PROGRAM GantryRobotMotion
VAR
	
	//Speed settings Adjustible from Visu
	MCJogVelocity		: LREAL := 100.0;
	MCAutoVelocity		: LREAL := 250.0;
	mxMCButtonManLowVelocity 	: BOOL;
	

	//Homing motion Settings
	MCHomingMode	: MC_HomingMode := MC_HomingMode.MC_DefaultHoming ;
	iMCXCaibratePos 	: INT := 8;
	iMCYCaibratePos 	: INT := 8;
	iMCZCaibratePos 	: INT := 8;

	//Manual motion Settings
	MCJogMode		: E_JogMode 	:= E_JogMode.MC_JOGMODE_CONTINOUS;
	MCJogAcceleration	: LREAL := 500.0;
	MCJogDeceleration	: LREAL := 1500.0;
	MCJogJerk			: LREAL := 800.0;
	
	//Auto Motion Settings
	MCAutoAcceleration	: LREAL := 500.0;
	MCAutoDeceleration	: LREAL := 500.0;
	MCAutoJerk			: LREAL := 500.0;
	
	
	//Safe Transport Position
	MCYSafePos : LREAL := 160.0;
	MCZLiftDist : LREAL := 50.0;


	//Connection NC to Physical Servo Drives
	MCXAxisRef: AXIS_REF;
	MCYAxisRef: AXIS_REF;
	MCZAxisRef: AXIS_REF;

	
	// Auto motion Settings
	MCBufferMode   	: MC_BufferMode := MC_BufferMode.MC_Aborting;	
	
	

	//General Condition flags
	mxGeneralCOntrolOk: BOOL;
	mxButtonGeneralControlOn: BOOL;
	mxButtonGeneralControlOff: BOOL;
	mxButtonStartAuto : BOOL;
	mxButtonStopAuto : BOOL;
	mxButtonAutoMode: BOOL;
	mxGeneralControlOn: BOOL;	
	mxManualMode: BOOL;	
	mxAutoMode: BOOL;
	mxLimSwOK: BOOL;
	mxMCPowerOn: BOOL;
	mxAxesStatusOk: BOOL;
	mxAutoOn: BOOL;
	fbTONpuls1: TON;
	fbTONpuls2: TON;
	mxControlOff: BOOL;
	
	//Motor Control Function Block
	//MC  Power
	fbMCXPower: MC_Power;	//X-Axis
	mxMCXButtonByPass: BOOL;
	mxMCXPowerOn: BOOL;	

	fbMCYPower: MC_Power;	//Y-Axis
	mxMCYButtonByPass: BOOL;
	mxMCYPowerOn: BOOL;	
	
	fbMCZPower: MC_Power;	//Z-Axis
	mxMCZButtonByPass: BOOL;
	mxMCZPowerOn: BOOL;	
	
	
	// MC Read Status
	fbMCXReadStatus	: MC_ReadStatus;
	MCXAxisStatus	: ST_AxisStatus;
	mxMCXAxisError	: BOOL;

	fbMCYReadStatus	: MC_ReadStatus;
	MCYAxisStatus	: ST_AxisStatus;
	mxMCYAxisError	: BOOL;

	fbMCZReadStatus	: MC_ReadStatus;
	MCZAxisStatus	: ST_AxisStatus;
	mxMCZAxisError	: BOOL;

	
	// MC Read Actual Position
	fbMCXReadActualPosition: MC_ReadActualPosition;
	fbMCYReadActualPosition: MC_ReadActualPosition;
	fbMCZReadActualPosition: MC_ReadActualPosition;
	MCActualPos: AbsPosition;	
		
	//MC Reset
	fbMCXReset: MC_Reset;	
	fbMCYReset: MC_Reset;	
	fbMCZReset: MC_Reset;	
	mxButtonResetError:BOOL;

	//MC Homing 
	fbMCXHome: MC_Home;			//X-axis
	mxMCXButtonHoming: BOOL;
	mxMCXHomingDone: BOOL;	
	
	fbMCYHome: MC_Home;			//Y-axis
	mxMCYButtonHoming: BOOL;
	mxMCYHomingDone: BOOL;	
	
	fbMCZHome: MC_Home;			//Z-axis
	mxMCZButtonHoming: BOOL;
	mxMCZHomingDone: BOOL;	
	mxHomingDone: BOOL;	
	
	//MC Jog
	fbMCXJog: MC_Jog;			//X-Axis
	mxMCXButtonJogFWD: BOOL;
	mxMCXButtonJogBWD: BOOL;
	
	fbMCYJog: MC_Jog;			//Y-Axis
	mxMCYButtonJogFWD: BOOL;
	mxMCYButtonJogBWD: BOOL;
	
	fbMCZJog: MC_Jog;			//Z-Axis
	mxMCZButtonJogFWD: BOOL;
	mxMCZButtonJogBWD: BOOL;
	
	
	//MC Move Absolute Position	(Auto Sequence)
	fbMCXMoveAbsolute: MC_MoveAbsolute;		//X-Axis
	mxMCXMoveAbs: BOOL;
	MCXMovAbsPos: LREAL;
	MCXMoveAbsVel: LREAL;
	MCXMoveAbsACC: LREAL;
	MCXMoveAbsDec: LREAL;
	MCXMoveAbsJerk: LREAL;
	mxMCXMoveAbsDone: BOOL;

	//MC Move Absolute Position
	fbMCYMoveAbsolute: MC_MoveAbsolute;  	//Y-Axis
	mxMCYMoveAbs: BOOL;
	MCYMovAbsPos: LREAL;
	MCYMoveAbsVel: LREAL;
	MCYMoveAbsACC: LREAL;
	MCYMoveAbsDec: LREAL;
	MCYMoveAbsJerk: LREAL;
	mxMCYMoveAbsDone: BOOL;
	
	fbMCXHalt: MC_Halt;
	fbMCYHalt: MC_Halt;
	fbMCZHalt: MC_Halt;
	

	//MC Move Absolute Position
	fbMCZMoveAbsolute: MC_MoveAbsolute;		//Z-Axis
	mxMCZMoveAbs: BOOL;
	MCZMovAbsPos: LREAL;
	MCZMoveAbsVel: LREAL;
	MCZMoveAbsACC: LREAL;
	MCZMoveAbsDec: LREAL;
	MCZMoveAbsJerk: LREAL;
	mxMCZMoveAbsDone: BOOL;
	
	//Modify Position
	ModPos	: AbsPosition;
	ModPosStation: INT := 1;
	ModPosLocation:INT := 1;
	mxButtonModPosExecute : BOOL;
	mxButtonSavePos : BOOL;
	fbTONButtonModPosExecute : TON;
	mxButtonReadFile: BOOL;
	mxReminderToSave : BOOL;
	
	
	// Gripper	
	mxTogleGripper : BOOL;
	fbTONGripperOn: TON;
	fbTONGripperOff: TON;	
	
	//Auto Sequence
	iSequence: INT; 
	arrAbsPosition: ARRAY[1..4, 1..9] OF AbsPosition;	//Station 100-400 Place 1 to 9
	mxButtonGoToModPos : BOOL;
	strStatusText : STRING;
	
	
	//File handling AbsPositions XYZ
	fbFileOpen    			: FB_FileOpen;
    fbFileRead              : FB_FileRead;
    fbFileWrite             : FB_FileWrite;
    fbFileClose             : FB_FileClose;    
	hFile                   : UINT   := 0;
	mxFileOpen				: BOOL;
	mxFileRead				: BOOL;	
	mxFileWrite				: BOOL;
	mxFileClose				: BOOL;
	nFileOpenMode			: DWORD;
	mxMemSavePos: BOOL;
	mxMemReadFile: BOOL;
	fbTONFileTime: TON;

END_VAR
VAR // added by the converter: edge detectors and wires of the graphical bodies
    _rt1, _rt2, _rt3, _rt4, _rt5, _rt6, _rt7 : R_TRIG;
END_VAR

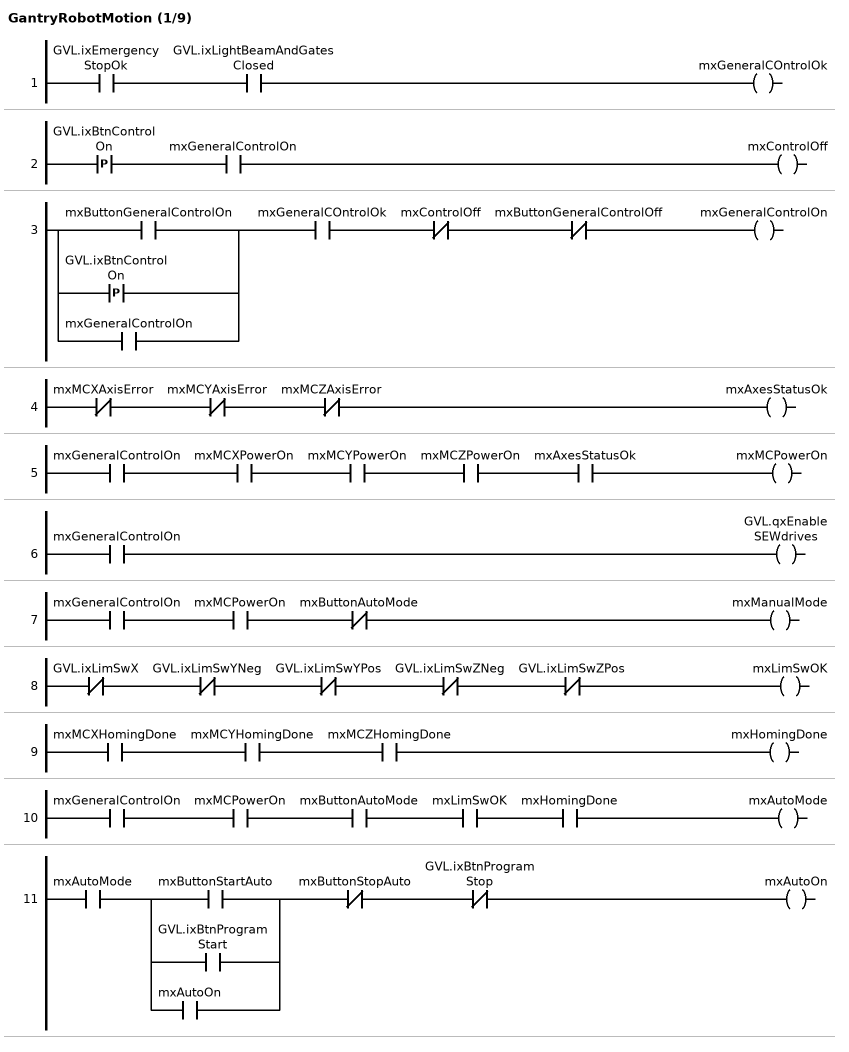
// NETWORK 1
mxGeneralCOntrolOk := GVL.ixEmergencyStopOk AND GVL.ixLightBeamAndGatesClosed;

// NETWORK 2
_rt1(CLK := GVL.ixBtnControlOn);
mxControlOff := _rt1.Q AND mxGeneralControlOn;

// NETWORK 3
_rt2(CLK := GVL.ixBtnControlOn);
mxGeneralControlOn := (mxButtonGeneralControlOn OR _rt2.Q OR mxGeneralControlOn) AND mxGeneralCOntrolOk AND NOT mxControlOff AND NOT mxButtonGeneralControlOff;

// NETWORK 4
mxAxesStatusOk := NOT mxMCXAxisError AND NOT mxMCYAxisError AND NOT mxMCZAxisError;

// NETWORK 5
mxMCPowerOn := mxGeneralControlOn AND mxMCXPowerOn AND mxMCYPowerOn AND mxMCZPowerOn AND mxAxesStatusOk;

// NETWORK 6
GVL.qxEnableSEWdrives := mxGeneralControlOn;

// NETWORK 7
mxManualMode := mxGeneralControlOn AND mxMCPowerOn AND NOT mxButtonAutoMode;

// NETWORK 8
mxLimSwOK := NOT GVL.ixLimSwX AND NOT GVL.ixLimSwYNeg AND NOT GVL.ixLimSwYPos AND NOT GVL.ixLimSwZNeg AND NOT GVL.ixLimSwZPos;

// NETWORK 9
mxHomingDone := mxMCXHomingDone AND mxMCYHomingDone AND mxMCZHomingDone;

// NETWORK 10
mxAutoMode := mxGeneralControlOn AND mxMCPowerOn AND mxButtonAutoMode AND mxLimSwOK AND mxHomingDone;

// NETWORK 11
mxAutoOn := mxAutoMode AND (mxButtonStartAuto OR GVL.ixBtnProgramStart OR mxAutoOn) AND NOT mxButtonStopAuto AND NOT GVL.ixBtnProgramStop;

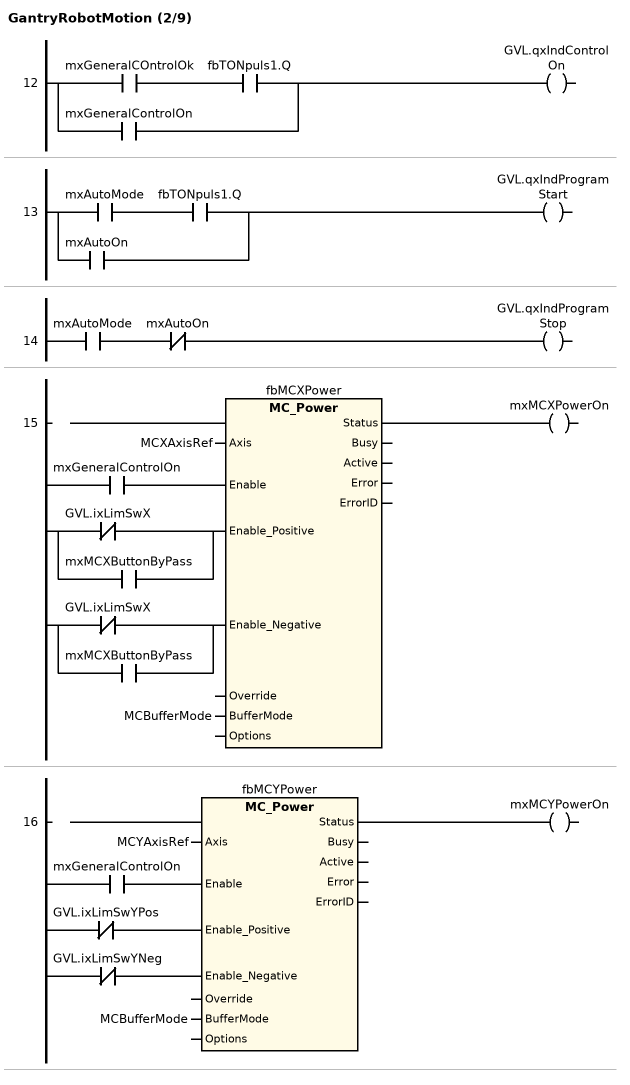
// NETWORK 12
GVL.qxIndControlOn := mxGeneralCOntrolOk AND fbTONpuls1.Q OR mxGeneralControlOn;

// NETWORK 13
GVL.qxIndProgramStart := mxAutoMode AND fbTONpuls1.Q OR mxAutoOn;

// NETWORK 14
GVL.qxIndProgramStop := mxAutoMode AND NOT mxAutoOn;

// NETWORK 15
fbMCXPower(
    Axis := MCXAxisRef,
    Enable := mxGeneralControlOn,
    Enable_Positive := NOT GVL.ixLimSwX OR mxMCXButtonByPass,
    Enable_Negative := NOT GVL.ixLimSwX OR mxMCXButtonByPass,
    BufferMode := MCBufferMode); // MC_Power
mxMCXPowerOn := fbMCXPower.Status;

// NETWORK 16
fbMCYPower(
    Axis := MCYAxisRef,
    Enable := mxGeneralControlOn,
    Enable_Positive := NOT GVL.ixLimSwYPos,
    Enable_Negative := NOT GVL.ixLimSwYNeg,
    BufferMode := MCBufferMode); // MC_Power
mxMCYPowerOn := fbMCYPower.Status;

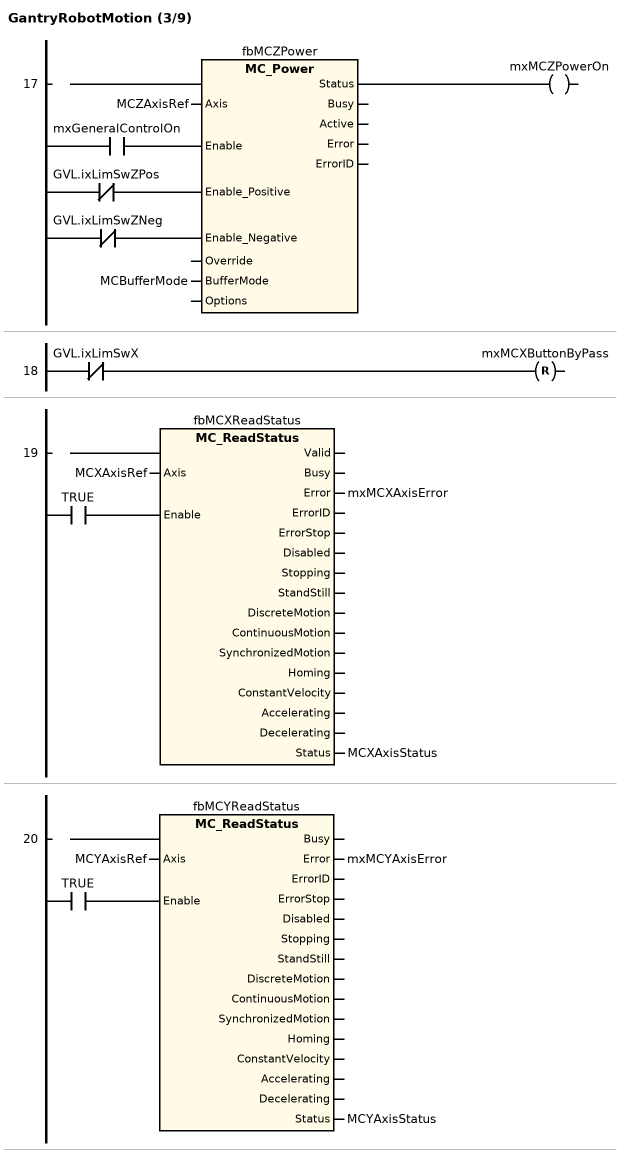
// NETWORK 17
fbMCZPower(
    Axis := MCZAxisRef,
    Enable := mxGeneralControlOn,
    Enable_Positive := NOT GVL.ixLimSwZPos,
    Enable_Negative := NOT GVL.ixLimSwZNeg,
    BufferMode := MCBufferMode); // MC_Power
mxMCZPowerOn := fbMCZPower.Status;

// NETWORK 18
mxMCXButtonByPass R= NOT GVL.ixLimSwX;

// NETWORK 19
fbMCXReadStatus(Axis := MCXAxisRef, Enable := TRUE, Error => mxMCXAxisError, Status => MCXAxisStatus); // MC_ReadStatus

// NETWORK 20
fbMCYReadStatus(Axis := MCYAxisRef, Enable := TRUE, Error => mxMCYAxisError, Status => MCYAxisStatus); // MC_ReadStatus

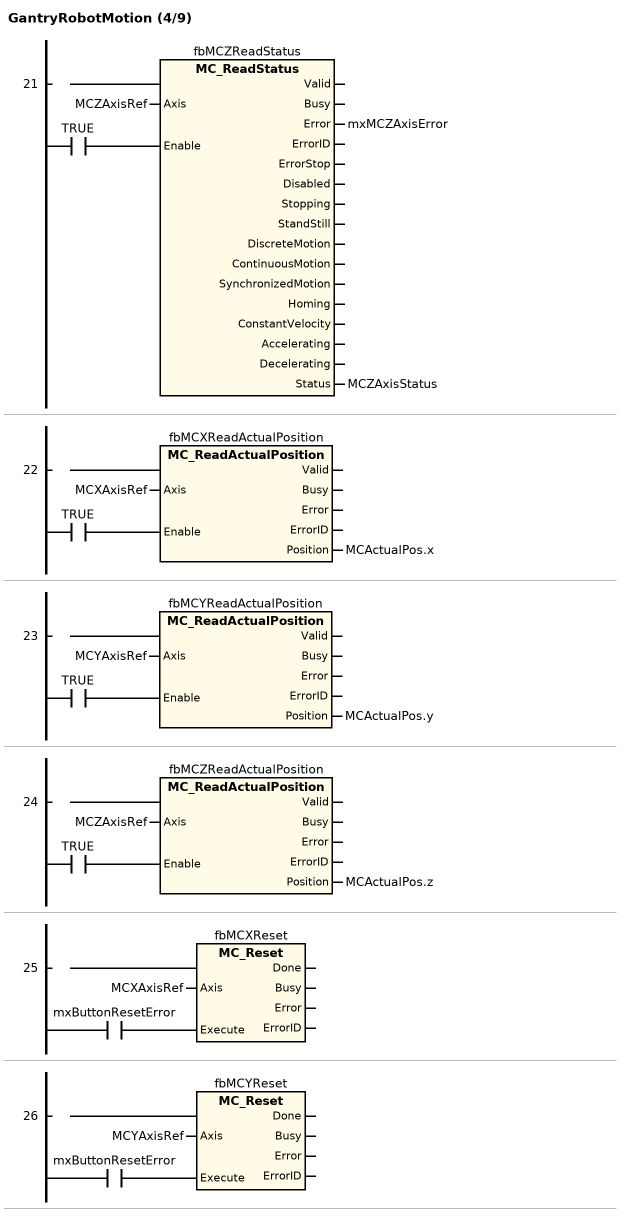
// NETWORK 21
fbMCZReadStatus(Axis := MCZAxisRef, Enable := TRUE, Error => mxMCZAxisError, Status => MCZAxisStatus); // MC_ReadStatus

// NETWORK 22
fbMCXReadActualPosition(Axis := MCXAxisRef, Enable := TRUE, Position => MCActualPos.x); // MC_ReadActualPosition

// NETWORK 23
fbMCYReadActualPosition(Axis := MCYAxisRef, Enable := TRUE, Position => MCActualPos.y); // MC_ReadActualPosition

// NETWORK 24
fbMCZReadActualPosition(Axis := MCZAxisRef, Enable := TRUE, Position => MCActualPos.z); // MC_ReadActualPosition

// NETWORK 25
fbMCXReset(Axis := MCXAxisRef, Execute := mxButtonResetError); // MC_Reset

// NETWORK 26
fbMCYReset(Axis := MCYAxisRef, Execute := mxButtonResetError); // MC_Reset

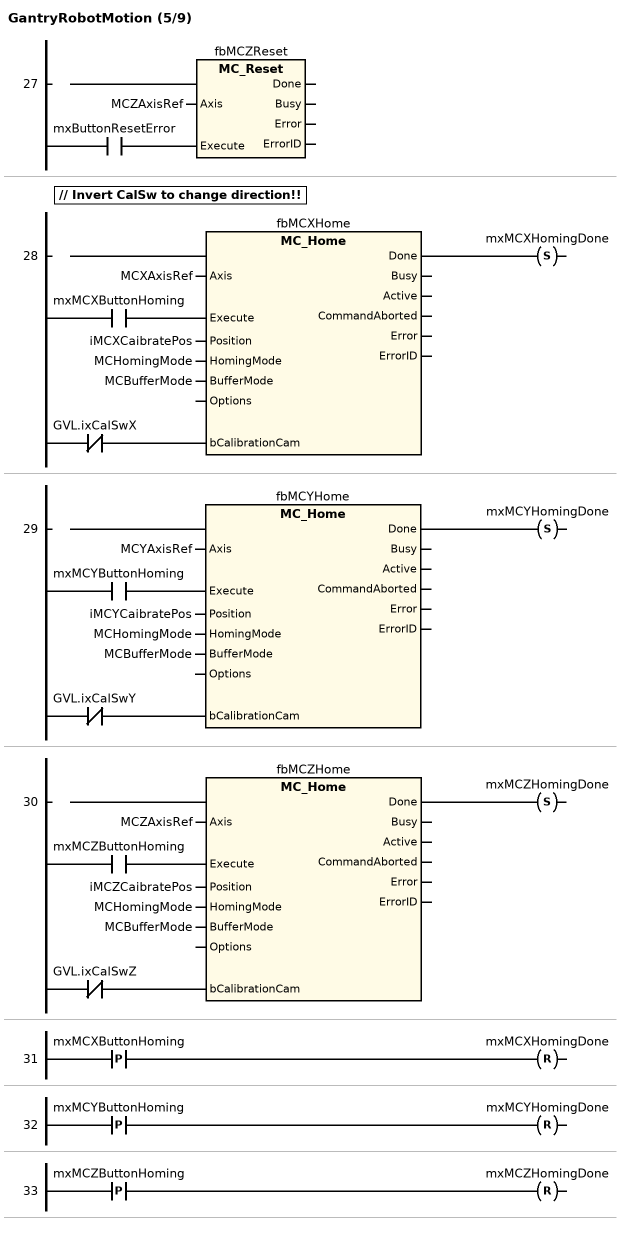
// NETWORK 27
fbMCZReset(Axis := MCZAxisRef, Execute := mxButtonResetError); // MC_Reset

// NETWORK 28
// label: // Invert CalSw to change direction!!
fbMCXHome(
    Axis := MCXAxisRef,
    Execute := mxMCXButtonHoming,
    Position := iMCXCaibratePos,
    HomingMode := MCHomingMode,
    BufferMode := MCBufferMode,
    bCalibrationCam := NOT GVL.ixCalSwX); // MC_Home
mxMCXHomingDone S= fbMCXHome.Done;

// NETWORK 29
fbMCYHome(
    Axis := MCYAxisRef,
    Execute := mxMCYButtonHoming,
    Position := iMCYCaibratePos,
    HomingMode := MCHomingMode,
    BufferMode := MCBufferMode,
    bCalibrationCam := NOT GVL.ixCalSwY); // MC_Home
mxMCYHomingDone S= fbMCYHome.Done;

// NETWORK 30
fbMCZHome(
    Axis := MCZAxisRef,
    Execute := mxMCZButtonHoming,
    Position := iMCZCaibratePos,
    HomingMode := MCHomingMode,
    BufferMode := MCBufferMode,
    bCalibrationCam := NOT GVL.ixCalSwZ); // MC_Home
mxMCZHomingDone S= fbMCZHome.Done;

// NETWORK 31
_rt3(CLK := mxMCXButtonHoming);
mxMCXHomingDone R= _rt3.Q;

// NETWORK 32
_rt4(CLK := mxMCYButtonHoming);
mxMCYHomingDone R= _rt4.Q;

// NETWORK 33
_rt5(CLK := mxMCZButtonHoming);
mxMCZHomingDone R= _rt5.Q;

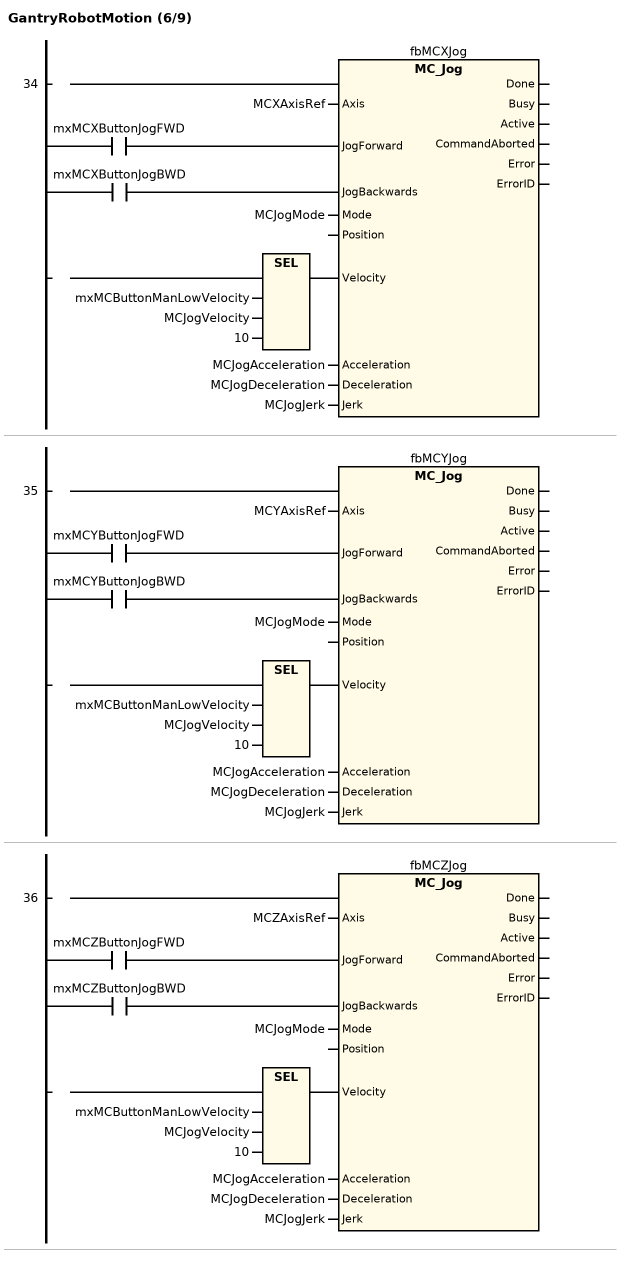
// NETWORK 34
fbMCXJog(
    Axis := MCXAxisRef,
    JogForward := mxMCXButtonJogFWD,
    JogBackwards := mxMCXButtonJogBWD,
    Mode := MCJogMode,
    Velocity := SEL(mxMCButtonManLowVelocity, MCJogVelocity, 10),
    Acceleration := MCJogAcceleration,
    Deceleration := MCJogDeceleration,
    Jerk := MCJogJerk); // MC_Jog

// NETWORK 35
fbMCYJog(
    Axis := MCYAxisRef,
    JogForward := mxMCYButtonJogFWD,
    JogBackwards := mxMCYButtonJogBWD,
    Mode := MCJogMode,
    Velocity := SEL(mxMCButtonManLowVelocity, MCJogVelocity, 10),
    Acceleration := MCJogAcceleration,
    Deceleration := MCJogDeceleration,
    Jerk := MCJogJerk); // MC_Jog

// NETWORK 36
fbMCZJog(
    Axis := MCZAxisRef,
    JogForward := mxMCZButtonJogFWD,
    JogBackwards := mxMCZButtonJogBWD,
    Mode := MCJogMode,
    Velocity := SEL(mxMCButtonManLowVelocity, MCJogVelocity, 10),
    Acceleration := MCJogAcceleration,
    Deceleration := MCJogDeceleration,
    Jerk := MCJogJerk); // MC_Jog

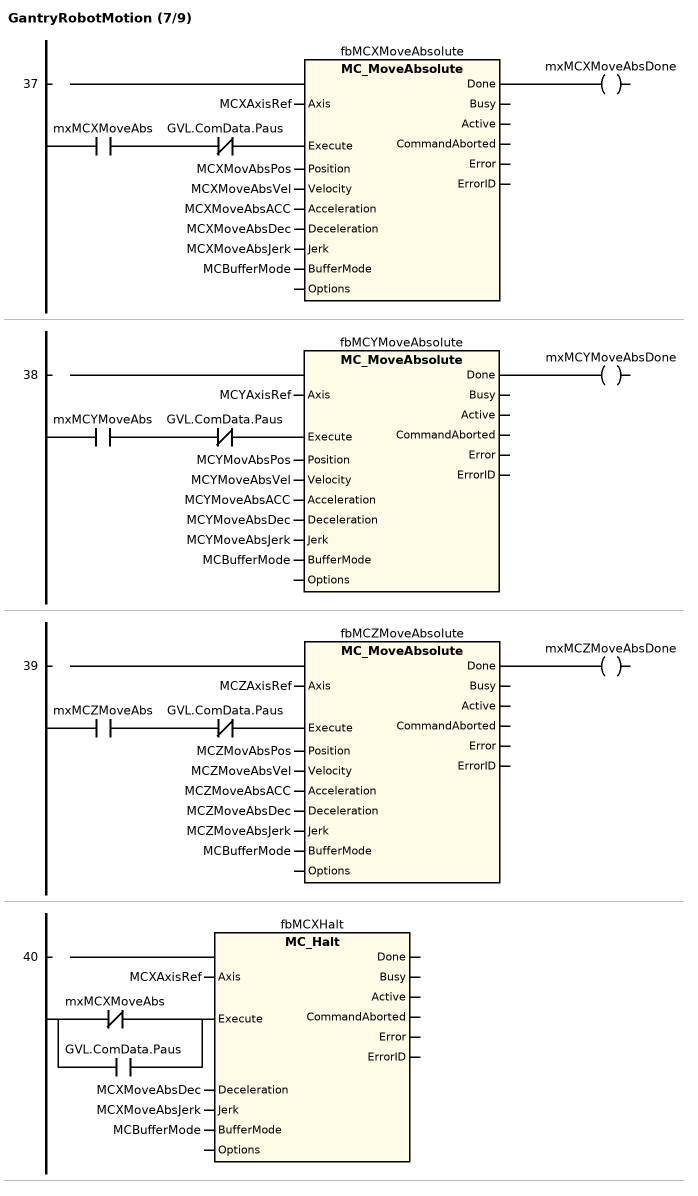
// NETWORK 37
fbMCXMoveAbsolute(
    Axis := MCXAxisRef,
    Execute := mxMCXMoveAbs AND NOT GVL.ComData.Paus,
    Position := MCXMovAbsPos,
    Velocity := MCXMoveAbsVel,
    Acceleration := MCXMoveAbsACC,
    Deceleration := MCXMoveAbsDec,
    Jerk := MCXMoveAbsJerk,
    BufferMode := MCBufferMode); // MC_MoveAbsolute
mxMCXMoveAbsDone := fbMCXMoveAbsolute.Done;

// NETWORK 38
fbMCYMoveAbsolute(
    Axis := MCYAxisRef,
    Execute := mxMCYMoveAbs AND NOT GVL.ComData.Paus,
    Position := MCYMovAbsPos,
    Velocity := MCYMoveAbsVel,
    Acceleration := MCYMoveAbsACC,
    Deceleration := MCYMoveAbsDec,
    Jerk := MCYMoveAbsJerk,
    BufferMode := MCBufferMode); // MC_MoveAbsolute
mxMCYMoveAbsDone := fbMCYMoveAbsolute.Done;

// NETWORK 39
fbMCZMoveAbsolute(
    Axis := MCZAxisRef,
    Execute := mxMCZMoveAbs AND NOT GVL.ComData.Paus,
    Position := MCZMovAbsPos,
    Velocity := MCZMoveAbsVel,
    Acceleration := MCZMoveAbsACC,
    Deceleration := MCZMoveAbsDec,
    Jerk := MCZMoveAbsJerk,
    BufferMode := MCBufferMode); // MC_MoveAbsolute
mxMCZMoveAbsDone := fbMCZMoveAbsolute.Done;

// NETWORK 40
fbMCXHalt(
    Axis := MCXAxisRef,
    Execute := NOT mxMCXMoveAbs OR GVL.ComData.Paus,
    Deceleration := MCXMoveAbsDec,
    Jerk := MCXMoveAbsJerk,
    BufferMode := MCBufferMode); // MC_Halt

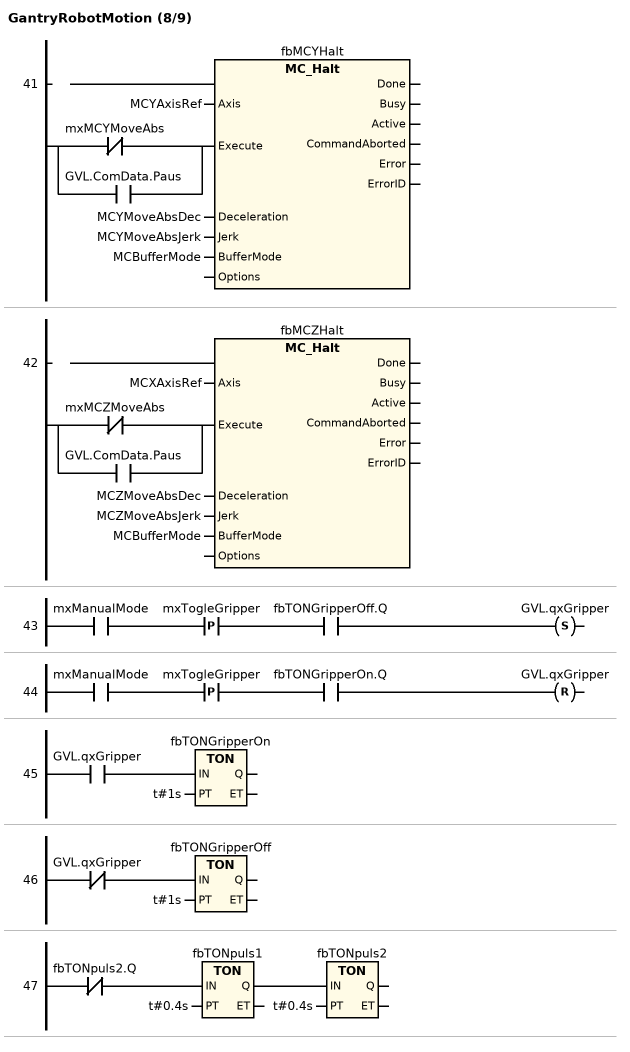
// NETWORK 41
fbMCYHalt(
    Axis := MCYAxisRef,
    Execute := NOT mxMCYMoveAbs OR GVL.ComData.Paus,
    Deceleration := MCYMoveAbsDec,
    Jerk := MCYMoveAbsJerk,
    BufferMode := MCBufferMode); // MC_Halt

// NETWORK 42
fbMCZHalt(
    Axis := MCXAxisRef,
    Execute := NOT mxMCZMoveAbs OR GVL.ComData.Paus,
    Deceleration := MCZMoveAbsDec,
    Jerk := MCZMoveAbsJerk,
    BufferMode := MCBufferMode); // MC_Halt

// NETWORK 43
_rt6(CLK := mxTogleGripper);
GVL.qxGripper S= mxManualMode AND _rt6.Q AND fbTONGripperOff.Q;

// NETWORK 44
_rt7(CLK := mxTogleGripper);
GVL.qxGripper R= mxManualMode AND _rt7.Q AND fbTONGripperOn.Q;

// NETWORK 45
fbTONGripperOn(IN := GVL.qxGripper, PT := t#1s); // TON

// NETWORK 46
fbTONGripperOff(IN := NOT GVL.qxGripper, PT := t#1s); // TON

// NETWORK 47
fbTONpuls1(IN := NOT fbTONpuls2.Q, PT := t#0.4s); // TON
fbTONpuls2(IN := fbTONpuls1.Q, PT := t#0.4s); // TON

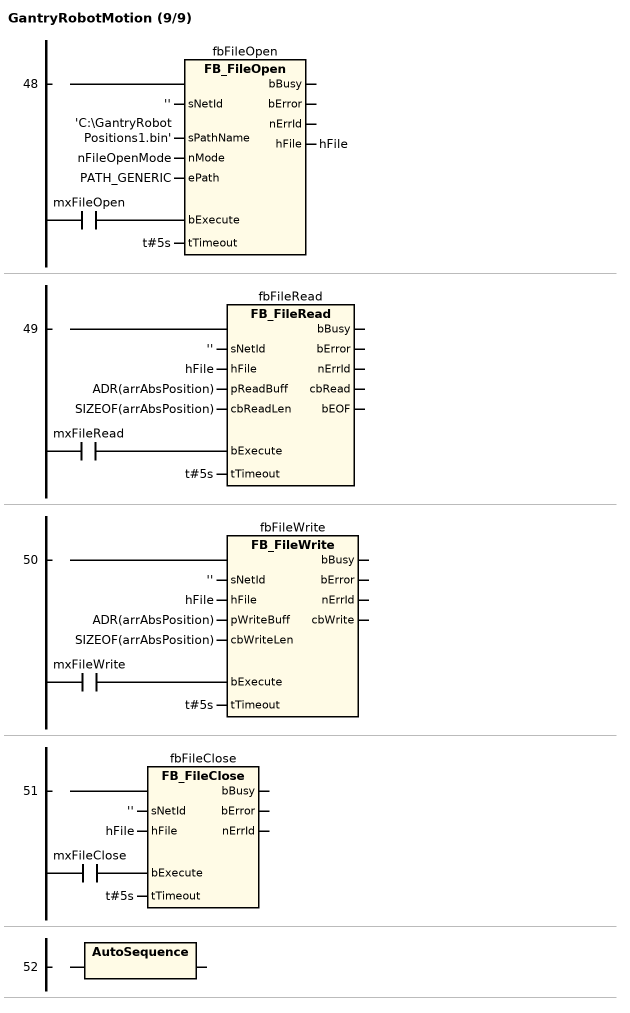
// NETWORK 48
fbFileOpen(
    sNetId := '',
    sPathName := 'C:\GantryRobotPositions1.bin',
    nMode := nFileOpenMode,
    ePath := PATH_GENERIC,
    bExecute := mxFileOpen,
    tTimeout := t#5s,
    hFile => hFile); // FB_FileOpen

// NETWORK 49
fbFileRead(
    sNetId := '',
    hFile := hFile,
    pReadBuff := ADR(arrAbsPosition),
    cbReadLen := SIZEOF(arrAbsPosition),
    bExecute := mxFileRead,
    tTimeout := t#5s); // FB_FileRead

// NETWORK 50
fbFileWrite(
    sNetId := '',
    hFile := hFile,
    pWriteBuff := ADR(arrAbsPosition),
    cbWriteLen := SIZEOF(arrAbsPosition),
    bExecute := mxFileWrite,
    tTimeout := t#5s); // FB_FileWrite

// NETWORK 51
fbFileClose(sNetId := '', hFile := hFile, bExecute := mxFileClose, tTimeout := t#5s); // FB_FileClose

// NETWORK 52
AutoSequence();

ACTION AutoSequence:


// Min Max Check Speed
IF MCJogVelocity > 250 THEN
	MCJogVelocity := 250;
END_IF
IF MCJogVelocity < 5 THEN
	MCJogVelocity := 5;
END_IF

IF MCAutoVelocity > 1000 THEN
	MCAutoVelocity := 1000;
END_IF
IF MCAutoVelocity < 100 THEN
	MCAutoVelocity := 100;
END_IF

	
// Copy status to function block interface
GVL.ComData.Status 		:= strStatusText;
GVL.ComData.ManualMode	:= mxManualMode;
GVL.ComData.Auto 		:= mxAutoOn;



CASE iSequence OF
	0:	// Init variable and read position file
		mxMCXMoveAbs := FALSE;
		mxMCYMoveAbs := FALSE;
		mxMCZMoveAbs := FALSE;
		fbTONButtonModPosExecute.PT := T#2S;
		fbTONButtonModPosExecute.IN := FALSE;
		fbTONButtonModPosExecute();

	
        // Open Gantry Robot Positions File for Read
		strStatusText := 'Reading Gantry Robot Position File'; 
		nFileOpenMode := FOPEN_MODEREAD OR FOPEN_MODEBINARY;
		mxFileOpen  := FALSE;
		mxFileRead  := FALSE;
		mxFileWrite := FALSE;
		mxFileClose := FALSE;	
		iSequence := 1;
		fbTONFileTime.IN := FALSE;
		fbTONFileTime.PT := T#3S;
		fbTONFileTime();
		
	
	1: // Wait for Opening of Gantry Robot Positions file and Check Errors
		fbTONFileTime.IN := TRUE;
		fbTONFileTime();
		mxFileOpen  := fbTONFileTime.q;
		IF mxFileOpen AND hFile > 0 AND NOT fbFileOpen.bBusy AND NOT fbFileOpen.bError THEN
			iSequence := 2;
		END_IF

	
	2:  // Read in Gantry Robot Positions File  to array of positions
		mxFileOpen  := FALSE;
		mxFileRead 	:= TRUE;
		iSequence := 3;		

			
	3:  // Wait for read Gantry Robot Positions File
		IF NOT fbFileRead.bBusy AND NOT fbFileRead.bError AND fbFileRead.cbRead = SIZEOF(arrAbsPosition) THEN
			iSequence := 4;
		END_IF
		

	4: // Close Gantry Robot Positions File
		mxFileRead  := FALSE;
		mxFileClose := TRUE;		
		strStatusText := 'Gantry Robot Position File Readed';		
		iSequence := 10;


	(* Write file *)
	5:  // Open Gantry Robot Positions Text File for Write
		strStatusText := 'Writing Gantry Robot Position File'; 
		nFileOpenMode := FOPEN_MODEWRITE OR FOPEN_MODEBINARY;
		mxFileOpen  := FALSE;
		mxFileRead  := FALSE;
		mxFileWrite := FALSE;
		mxFileClose := FALSE;	
		fbTONFileTime.IN := FALSE;
		fbTONFileTime.PT := T#3S;
		fbTONFileTime();
		iSequence := 6;
		
	
	6: // Wait for Opening of Gantry Robot Positions File and Check Errors
		fbTONFileTime.IN := TRUE;
		fbTONFileTime();
		mxFileOpen  := fbTONFileTime.Q;
		IF mxFileOpen AND hFile > 0 AND NOT fbFileOpen.bBusy AND NOT fbFileOpen.bError THEN
			iSequence := 7;
		END_IF
	
	
	7:  // Write Gantry Robot Positions File from array of positions
		mxFileOpen  := FALSE;
		mxFileWrite := TRUE;
		iSequence := 8;		

			
	8:	// Wait for Write Gantry Robot Positions File
		IF NOT fbFileWrite.bBusy AND NOT fbFileWrite.bError AND fbFileWrite.cbWrite = SIZEOF(arrAbsPosition) THEN
			iSequence := 9;
		END_IF


	9: 	// Close Gantry Robot Positions File
		strStatusText := 'Gantry Robot Positions Saved'; 		
		mxFileWrite  := FALSE;
		mxFileClose := TRUE;		
		iSequence := 10;

		
	10: // ********* Wait for auto or Modify Position, Save to file and status in Manual mode  ***************
	
		//Status text
		IF NOT GVL.ixEmergencyStopOk THEN
			strStatusText := 'Emergency Stop Activated';
		ELSIF NOT GVL.ixLightBeamAndGatesClosed THEN
			strStatusText := 'Safety Stop (Gate) Activated';
		ELSIF mxGeneralCOntrolOk AND NOT mxGeneralControlOn THEN
			strStatusText := 'Ready for General Power';
		ELSIF mxGeneralControlOn AND NOT mxMCPowerOn THEN
			strStatusText := 'Servo Drives Fault';
		ELSIF mxManualMode THEN
			strStatusText := 'Manual Mode OK';	
		ELSIF mxButtonAutoMode AND NOT mxLimSwOK THEN
			strStatusText := 'End Limit Switch Activated';
		ELSIF mxButtonAutoMode AND NOT mxHomingDone THEN
			strStatusText := 'Axes Not in reference (Run Homing)';
		ELSIF mxButtonAutoMode AND NOT mxAutoOn THEN
			strStatusText := 'Ready for Start Auto';
		ELSIF mxAutoOn THEN
			strStatusText := 'Ready for Order Auto';
		END_IF
		
					
		// Run in auto mode
		IF mxAutoOn THEN
			iSequence := 100;
		END_IF
	
		GVL.ComData.AckPickPosition := 0;
		GVL.ComData.AckPickStation := 0;
		GVL.ComData.AckLeavePosition := 0;
		GVL.ComData.AckLeaveStation := 0;
		
	
		// Move to "Modify Position" in HMI selected Robot Station and Storage Loacation 
		IF mxButtonGoToModPos AND mxManualMode AND mxHomingDone THEN //Manual Mode
			iSequence := 20;	
		END_IF
		
		// Modify position
		IF  mxButtonModPosExecute AND mxManualMode THEN
			arrAbsPosition[ModPosStation, ModPosLocation] := MCActualPos;
			mxReminderToSave := TRUE;
		END_IF
		
		// Save Position
		IF mxButtonSavePos AND NOT mxMemSavePos THEN
			iSequence := 5; //Write file
			mxReminderToSave := FALSE;
		END_IF
		mxMemSavePos := mxButtonSavePos;
		
		// Read file (UnDo)
		IF mxButtonReadFile AND NOT mxMemReadFile THEN
			iSequence := 0; //Read file
			mxReminderToSave := FALSE;
		END_IF
		mxMemReadFile := mxButtonReadFile;
		
		// Auto motion	
		IF mxAutoOn THEN
			IF GVL.ComData.LeavePosition = 0 
				AND GVL.ComData.LeaveStation = 0 
					AND GVL.ComData.PickPosition = 0 
						AND GVL.ComData.PickStation = 0 	THEN
				iSequence := 100;		//Auto mode					
			ELSE
				strStatusText := 'Clear Old Order';
			END_IF;
		END_IF
		

	
	20: 	//Init Speed Acc Dec Jerk for Manual Mode ( Goto ModPos) 
		MCXMoveAbsVel	:= MCJogVelocity ;
		MCXMoveAbsACC	:= MCJogAcceleration;
		MCXMoveAbsDec	:= MCJogDeceleration;
		MCXMoveAbsJerk	:= MCJogJerk;

		MCYMoveAbsVel	:= MCJogVelocity ;
		MCYMoveAbsACC	:= MCJogAcceleration;
		MCYMoveAbsDec	:= MCJogDeceleration;
		MCYMoveAbsJerk	:= MCJogJerk;

		MCZMoveAbsVel	:= MCJogVelocity ;
		MCZMoveAbsACC	:= MCJogAcceleration;
		MCZMoveAbsDec	:= MCJogDeceleration;
		MCZMoveAbsJerk	:= MCJogJerk;
		strStatusText := 'Moving to Modify Position';

		iSequence := 30;
		
		
	30:		// Move Y to safe position in the passage ( Goto ModPos)
		MCYMovAbsPos	:= MCYSafePos;
		mxMCYMoveAbs	:= TRUE;
		
		IF mxMCYMoveAbsDone THEN
			mxMCYMoveAbs := FALSE;
			iSequence := 40;
		END_IF
		
 		IF NOT mxButtonGoToModPos OR NOT mxManualMode THEN
			mxMCYMoveAbs:= FALSE;
			iSequence := 10;
		END_IF

		
	40:		// Move X And Z to Above Loacation ( Goto ModPos)
		MCXMovAbsPos	:= arrAbsPosition[ ModPosStation, ModPosLocation].x;
		mxMCXMoveAbs	:= TRUE;

		MCZMovAbsPos	:= arrAbsPosition[ ModPosStation, ModPosLocation].z - MCZLiftDist;
		mxMCZMoveAbs	:= TRUE;

	
		IF mxMCXMoveAbsDone AND mxMCZMoveAbsDone THEN
			mxMCXMoveAbs:= FALSE;
			mxMCZMoveAbs:= FALSE;
			iSequence 	:= 50;
		END_IF
		
		IF NOT mxButtonGoToModPos OR NOT mxManualMode THEN
			mxMCXMoveAbs:= FALSE;
			mxMCZMoveAbs:= FALSE;
			iSequence 	:= 10;
		END_IF
	
		
	50:		// Move Y in to storage ( Goto ModPos)
		MCYMovAbsPos		:= arrAbsPosition[ ModPosStation, ModPosLocation].y;
		mxMCYMoveAbs		:= TRUE;
		
		IF mxMCYMoveAbsDone THEN
			mxMCYMoveAbs 	:= FALSE;
			iSequence 		:= 60;
		END_IF
		
		IF NOT mxButtonGoToModPos OR NOT mxManualMode THEN
			mxMCYMoveAbs	:= FALSE;
			iSequence 		:= 0;
		END_IF
		
		
	60:		// Move Z down to storage ( Go to ModPos)	
		MCZMovAbsPos	:= arrAbsPosition[ ModPosStation, ModPosLocation].z;
		mxMCZMoveAbs	:= TRUE;
		
		IF mxMCYMoveAbsDone THEN
			strStatusText := 'In Modify Position';
		END_IF
		
		IF NOT mxButtonGoToModPos OR NOT mxManualMode THEN
			mxMCZMoveAbs:= FALSE;
			iSequence 	:= 10;
		END_IF

	
	
	100: 	// Init Auto speed acc and jerk ( Auto)
		MCXMoveAbsVel	:= MCAutoVelocity ;
		MCXMoveAbsACC	:= MCAutoAcceleration;
		MCXMoveAbsDec	:= MCAutoDeceleration;
		MCXMoveAbsJerk	:= MCAutoJerk;

		MCYMoveAbsVel	:= MCAutoVelocity ;
		MCYMoveAbsACC	:= MCAutoAcceleration;
		MCYMoveAbsDec	:= MCAutoDeceleration;
		MCYMoveAbsJerk	:= MCAutoJerk;

		MCZMoveAbsVel	:= MCAutoVelocity ;
		MCZMoveAbsACC	:= MCAutoAcceleration;
		MCZMoveAbsDec	:= MCAutoDeceleration;
		MCZMoveAbsJerk	:= MCAutoJerk;

		iSequence 		:= 110;

		
	110:  // Move Y to safe position in the passage ( Auto)
		MCYMovAbsPos	:= MCYSafePos;
		mxMCYMoveAbs	:= TRUE;
		strStatusText := 'Moving Y-axis to Transport Position';
	
		IF mxMCYMoveAbsDone THEN
			mxMCYMoveAbs := FALSE;
			iSequence := 120;
		END_IF
		
		IF NOT mxAutoOn THEN
			mxMCYMoveAbs:= FALSE;
			iSequence := 10;
		END_IF	

	
	120: 	// Ready for order  ( Auto)
		strStatusText := 'Ready for Order';
		iSequence := 130;

		IF NOT mxAutoOn THEN
			iSequence := 10;
		END_IF
		
		
	130:  	// *************************************** Wait for order ( Auto)  **************************************************
		IF GVL.ComData.PickPosition > 0	AND GVL.ComData.PickStation > 0 THEN
			GVL.ComData.AckPickPosition	:= 	GVL.ComData.PickPosition; //Acknowledge to function block
			GVL.ComData.AckPickStation	:= 	GVL.ComData.PickStation;
			iSequence := 200;
		END_IF		

		IF GVL.ComData.LeavePosition > 0 AND GVL.ComData.LeaveStation > 0 THEN
			GVL.ComData.AckLeavePosition	:= 	GVL.ComData.LeavePosition;
			GVL.ComData.AckLeaveStation		:= 	GVL.ComData.LeaveStation;
			iSequence := 300;
		END_IF
		

		IF NOT mxAutoOn THEN
			iSequence := 10;
		END_IF
		

	(* Auto Pickup sequence *)
	200: 	//Check Order (Auto Pickup) 	
		IF  GVL.ComData.PickPosition > 0 
			AND GVL.ComData.PickPosition <=9 
				AND GVL.ComData.PickStation > 0 
					AND GVL.ComData.PickStation <= 4 THEN
			iSequence := 210;
		ELSE
			strStatusText := 'Wrong Pickup Order Address';
			IF GVL.ComData.PickPosition = 0 AND GVL.ComData.PickStation = 0 THEN
				iSequence := 10;
			END_IF
		END_IF

		IF NOT mxAutoOn OR GVL.ComData.PickPosition = 0 OR	 GVL.ComData.PickStation = 0 THEN
			iSequence := 10;
		END_IF


	210:	// Move X And Z to Above and Outside the Loacation ( Auto Pickup)

		MCXMovAbsPos	:=  arrAbsPosition[ GVL.ComData.PickStation, GVL.ComData.PickPosition].x;
		mxMCXMoveAbs	:= TRUE;

		MCZMovAbsPos	:= arrAbsPosition[ GVL.ComData.PickStation, GVL.ComData.PickPosition].z - MCZLiftDist;
		mxMCZMoveAbs	:= TRUE;
		
		GVL.qxGripper := FALSE;
		strStatusText := 'Moving to Pickup Pallet';
		

		IF mxMCXMoveAbsDone AND mxMCZMoveAbsDone THEN
			mxMCXMoveAbs:= FALSE;
			mxMCZMoveAbs:= FALSE;
			iSequence 	:= 220;
		END_IF

		
		IF NOT mxAutoOn OR GVL.ComData.PickPosition = 0 OR	 GVL.ComData.PickStation = 0 THEN
			mxMCXMoveAbs:= FALSE;
			mxMCZMoveAbs:= FALSE;
			iSequence 	:= 10;
		END_IF
	
		
	220:	// Move Y in to storage (  Auto Pickup)
		MCYMovAbsPos		:=  arrAbsPosition[ GVL.ComData.PickStation, GVL.ComData.PickPosition].y;
		mxMCYMoveAbs		:= TRUE;
	
		IF mxMCYMoveAbsDone THEN
			mxMCYMoveAbs 	:= FALSE;
			iSequence 		:= 230;
		END_IF
		
		IF NOT mxAutoOn OR GVL.ComData.PickPosition = 0 OR	 GVL.ComData.PickStation = 0 THEN
			mxMCYMoveAbs	:= FALSE;
			iSequence 		:= 10;
		END_IF
			
		
	230:	// Move Z down to storage ( Auto Pickup)	
		MCZMovAbsPos	:= arrAbsPosition[ GVL.ComData.PickStation, GVL.ComData.PickPosition].z;
		mxMCZMoveAbs	:= TRUE;
		GVL.qxGripper := FALSE;
		
		IF mxMCZMoveAbsDone THEN
			mxMCZMoveAbs:= FALSE;
			iSequence 	:= 240;				
		END_IF
		
		IF NOT mxAutoOn OR GVL.ComData.PickPosition = 0 OR	 GVL.ComData.PickStation = 0  THEN
			mxMCZMoveAbs:= FALSE;
			iSequence 	:= 10;
		END_IF
		
	
	240:	//Grip pallet ( Auto Pickup)	
		GVL.qxGripper 	:= TRUE;
		strStatusText := 'Gripping the Pallet';
		IF fbTONGripperOn.Q THEN
			iSequence := 250;
		END_IF 
		
		IF NOT mxAutoOn OR GVL.ComData.PickPosition = 0 OR	 GVL.ComData.PickStation = 0  THEN
			iSequence 	:= 10;
		END_IF
		
		
	250: 	// Move Z up above storage ( Auto Pickup)	
		MCZMovAbsPos	:= arrAbsPosition[ GVL.ComData.PickStation, GVL.ComData.PickPosition].z - MCZLiftDist;
		mxMCZMoveAbs	:= TRUE;
		strStatusText := 'Moving out with the Pallet';
		
		IF mxMCZMoveAbsDone THEN
			mxMCZMoveAbs:= FALSE;
			iSequence := 260;
		END_IF
		
		IF NOT mxAutoOn OR GVL.ComData.PickPosition = 0 OR	 GVL.ComData.PickStation = 0  THEN
			mxMCZMoveAbs:= FALSE;
			iSequence 	:= 10;
		END_IF
		
		
	260:  	// Move Y to transport position ( Auto Pickup)	
		MCYMovAbsPos	:= MCYSafePos;
		mxMCYMoveAbs	:= TRUE;
	
		IF mxMCYMoveAbsDone THEN
			mxMCYMoveAbs := FALSE;
			GVL.ComData.AckPickPosition := 0;
			GVL.ComData.AckPickStation := 0;
			iSequence := 270;
		END_IF		
		
		IF NOT mxAutoOn OR GVL.ComData.PickPosition = 0 OR	 GVL.ComData.PickStation = 0 THEN
			mxMCYMoveAbs:= FALSE;
			iSequence := 10;
		END_IF

	
	270: 	// Wait for clear order
		strStatusText := 'Pickup pallet Done, Clear the order';
		IF 	GVL.ComData.PickStation = 0 AND GVL.ComData.PickPosition = 0 THEN
			strStatusText := 'Ready for Leave Order';
			iSequence := 130;
		END_IF	
		
		IF NOT mxAutoOn THEN
			mxMCYMoveAbs:= FALSE;
			iSequence := 10;
		END_IF

		
	300:  // Check Order 	( Auto Leave)
		IF  GVL.ComData.LeavePosition > 0 
			AND GVL.ComData.LeavePosition <=9 
				AND GVL.ComData.LeaveStation > 0 
					AND GVL.ComData.LeaveStation <= 4 THEN
			iSequence := 310;
		ELSE
			strStatusText := 'Wrong Leave Order Address';
			IF GVL.ComData.LeavePosition = 0 AND GVL.ComData.LeaveStation = 0 THEN
				iSequence := 10;
			END_IF
		END_IF

		IF NOT mxAutoOn THEN
			iSequence := 10;
		END_IF

	310:	// Move X And Z to Above and Outside the Loacation ( Auto Leave)
		MCXMovAbsPos	:= arrAbsPosition[ GVL.ComData.LeaveStation, GVL.ComData.LeavePosition].x;
		mxMCXMoveAbs	:= TRUE;

		MCZMovAbsPos	:= arrAbsPosition[ GVL.ComData.LeaveStation, GVL.ComData.LeavePosition].z - MCZLiftDist;
		mxMCZMoveAbs	:= TRUE;
		strStatusText := 'Moving to Leave Pallet';

		IF mxMCXMoveAbsDone AND mxMCZMoveAbsDone THEN
			mxMCXMoveAbs:= FALSE;
			mxMCZMoveAbs:= FALSE;
			iSequence 	:= 320;
		END_IF
		
		IF NOT mxAutoOn OR GVL.ComData.LeavePosition = 0 OR	 GVL.ComData.LeaveStation = 0 THEN
			mxMCXMoveAbs:= FALSE;
			mxMCZMoveAbs:= FALSE;
			iSequence 	:= 10;
		END_IF
	
		
	320:	// Move Y in to storage (  Auto Leave)
		MCYMovAbsPos		:= arrAbsPosition[ GVL.ComData.LeaveStation, GVL.ComData.LeavePosition].y;
		mxMCYMoveAbs		:= TRUE;
	
		IF mxMCYMoveAbsDone THEN
			mxMCYMoveAbs 	:= FALSE;
			iSequence 		:= 330;
		END_IF
		
		IF NOT mxAutoOn OR GVL.ComData.LeavePosition = 0 OR	 GVL.ComData.LeaveStation = 0 THEN
			mxMCYMoveAbs	:= FALSE;
			iSequence 		:= 10;
		END_IF
			
		
	330:	// Move Z down to storage ( Auto Leave)	
		MCZMovAbsPos	:= arrAbsPosition[ GVL.ComData.LeaveStation, GVL.ComData.LeavePosition].z;
		mxMCZMoveAbs	:= TRUE;
		
		IF mxMCZMoveAbsDone THEN
			mxMCZMoveAbs:= FALSE;
			iSequence 	:= 340;				
		END_IF
		
		IF NOT mxAutoOn OR GVL.ComData.LeavePosition = 0 OR	 GVL.ComData.LeaveStation = 0  THEN
			mxMCZMoveAbs:= FALSE;
			iSequence 	:= 10;
		END_IF
		
		
	340: 	// Release Gripper ( Auto Leave)
		GVL.qxGripper 	:= FALSE;
		strStatusText := 'Ungriping the Pallet';
		IF fbTONGripperOff.Q THEN
			iSequence := 350;
		END_IF 
		
		IF NOT mxAutoOn OR GVL.ComData.LeavePosition = 0 OR	 GVL.ComData.LeaveStation = 0  THEN
			iSequence 	:= 0;
		END_IF
		
		
	350:	// Move Z up above storage ( Auto Leave)	
		MCZMovAbsPos	:= arrAbsPosition[ GVL.ComData.LeaveStation, GVL.ComData.LeavePosition].z - MCZLiftDist;
		mxMCZMoveAbs	:= TRUE;
		strStatusText := 'Moving up from storage';
		
		IF mxMCZMoveAbsDone AND fbTONGripperOff.Q THEN
			mxMCZMoveAbs := FALSE;
			iSequence 	 := 360;
		END_IF
		
		IF NOT mxAutoOn OR GVL.ComData.LeavePosition = 0 OR	 GVL.ComData.LeaveStation = 0  THEN
			mxMCZMoveAbs := FALSE;
			iSequence 	 := 10;
		END_IF
		
		
	360: 	// Move Y to transport position ( Auto Leave)	
		MCYMovAbsPos	:= MCYSafePos;
		mxMCYMoveAbs	:= TRUE;
		strStatusText 	:= 'Moving out from storage';
	
		IF mxMCYMoveAbsDone THEN
			mxMCYMoveAbs := FALSE;
			GVL.ComData.AckLeavePosition := 0;
			GVL.ComData.AckLeaveStation := 0;
			iSequence 	 := 370;
		END_IF		
		
		IF NOT mxAutoOn OR GVL.ComData.LeavePosition = 0 OR	 GVL.ComData.LeaveStation = 0 THEN
			mxMCYMoveAbs:= FALSE;
			iSequence := 10;
		END_IF

		
	370: 	// Wait for clear order
		strStatusText 	:= 'Leave pallet Done, Clear the order';
		IF 	GVL.ComData.LeaveStation = 0 AND GVL.ComData.LeavePosition = 0 THEN
			strStatusText := 'Ready for Order';
			iSequence := 130;
		END_IF	
		
		IF NOT mxAutoOn THEN
			mxMCYMoveAbs:= FALSE;
			iSequence := 10;
		END_IF

	
END_CASE
END_ACTION

END_PROGRAM

(* stored: Version 1.1.0.1, ProductVersion 3.1.4022.12
   POU GantryRobotMotion: Id {078411d6-07d1-4660-ba0c-7bcbd330848e}, SpecialFunc None
   Action AutoSequence: Id {ed9255ba-6efd-4f6f-9ed2-51c2a861641d} *)
